(* PLC project template_grafcet_FMS.project, CODESYS CODESYS V3.5 SP22 *)
(* stored: creationDateTime 2026-03-28T03:34:54.1557026, modificationDateTime 2026-03-28T03:28:33.2760948 *)

(* |=========================================================================| | TEMPLATE ORIENTATIVO PARA A CONSTRUÇÃO DO GRAFCET/SFC DO PROJETO FINAL | |=========================================================================| | Instruções: | | 1. Cada etapa representa um estado do seu processo no FMS; | | 2. Adicione novas etapas e transições conforme o seu projeto; | | 3. Nomeie as etapas e variáveis de forma descritiva; | | 4. Se preferir comente o que cada etapa faz (isso ajuda muito!!) | | 5. Ao finalizar: | | - Vá em "Projeto" -> "Exportar" -> "Exporta PLCOpenXML" | | - Escolha apenas o POU principal (PLC_PRG) | | - Salve como <nome_do_projeto>.xml | | 6. Faça o upload no site para validação | |=========================================================================| *)
{attribute 'do_checks_for_implicit_code'}
PROGRAM PLC_PRG
  VAR
    Start_Processo : BOOL := FALSE;  (* Inicia o processo *)
    Para_Processo : BOOL := FALSE;  (* Para o processo *)
    Etapa1_Ativa : BOOL := FALSE;  (* Variáveis de estado *)
    Etapa2_Ativa : BOOL := FALSE;
    Etapa3_Ativa : BOOL := FALSE;
    Transicao_1_2 : BOOL := FALSE;  (* Condição de transição *)
    Transicao_2_3 : BOOL := FALSE;
    Transicao_3_Init : BOOL := FALSE;
    Sensor_Y_Home : BOOL := FALSE;  (* Sensores e/ou atuadores *)
    Sensor_Z_Home : BOOL := FALSE;
    Sensor_Garra : BOOL := FALSE;
    Motor1 : BOOL := FALSE;
    Motor2 : BOOL := FALSE;
    Valvula1 : BOOL := FALSE;
    Timer_11 : BOOL := FALSE;  (* Timers simulados *)
    Timer_25 : BOOL := FALSE;
  END_VAR

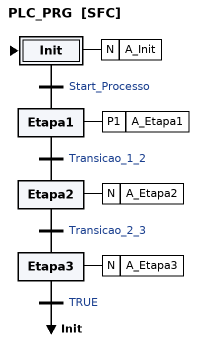
INITIAL_STEP Init:
  A_Init(N);
END_STEP
TRANSITION FROM Init TO Etapa1
  := Start_Processo;
END_TRANSITION
STEP Etapa1:
  A_Etapa1(P1);
END_STEP
TRANSITION FROM Etapa1 TO Etapa2
  := Transicao_1_2;
END_TRANSITION
STEP Etapa2:
  A_Etapa2(N);
END_STEP
TRANSITION FROM Etapa2 TO Etapa3
  := Transicao_2_3;
END_TRANSITION
STEP Etapa3:
  A_Etapa3(N);
END_STEP
TRANSITION FROM Etapa3 TO Init
  := TRUE;
END_TRANSITION

ACTION A_Etapa1:
                // STEP 1

Etapa1_Ativa := TRUE;

// Ação - movimentar eixo Y para a posição Home
// Insira lógica de acionamento se necessário

IF Sensor_Y_Home THEN
	Transicao_1_2 := TRUE;
END_IF
              
END_ACTION

ACTION A_Etapa2:
                // Step 2

Etapa2_Ativa := TRUE;

// Ação - Deslocar Eixo Z e confirmar a posição
// Inserir condição de avanço

IF Sensor_Z_Home THEN
	Transicao_2_3 := TRUE;
END_IF
              
END_ACTION

ACTION A_Init:
                // INICIALIZAÇÃO

Etapa1_Ativa := FALSE;
Etapa2_Ativa := FALSE;
Etapa3_Ativa := FALSE;
Transicao_1_2 := FALSE;
Transicao_2_3 := FALSE;
Transicao_3_Init := FALSE;
              
END_ACTION

ACTION A_Etapa3:
                // Step 3

Etapa3_Ativa := TRUE;

// Ação: Simular a operação do armazém, ex: garra para pegar o objeto

IF Timer_11 THEN
	Transicao_3_Init := TRUE;
END_IF

              
END_ACTION
END_PROGRAM
